// TIA Portal V18 export
DATA_BLOCK "Targets"   // DB23
{ S7_Optimized_Access := 'TRUE' }
VERSION : 0.1
// stored: AutoNumber true, DBAccessibleFromOPCUA true, IsOnlyStoredInLoadMemory false, IsRetainMemResEnabled false, IsWriteProtectedInAS false, MemoryReserve 100
   VAR RETAIN
      "A" : Array[1..10] of "typePositions";
   END_VAR
BEGIN
END_DATA_BLOCK
